{attribute addProperty BoxType "EL3773-0000-0016"}
{attribute addProperty Id "U3_SAMPLESAT %I*ARRAY [1..10] OF INT16020"}
{attribute addProperty CRC "3989497452"}
{attribute addProperty SizeInBites "160"}
{attribute addProperty SizeInBytes "20"}
TYPE L3_Voltage_Samples_EDCAE66C :
STRUCT
	{attribute addProperty Name "U3_SAMPLES"}
	U3_SAMPLES AT %I* : ARRAY [1..10] OF INT;
END_STRUCT
END_TYPE

(* stored: Version 1.2.0.0, ProductVersion 3.1.4024.9
   DUT L3_Voltage_Samples_EDCAE66C: Id {da87edf6-b991-42a6-b5e5-0fe67a829ffe} *)
